(* PLC project  *)

PROGRAM Sensor

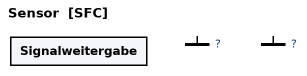
INITIAL_STEP Sensor bereit:
END_STEP
STEP Signalweitergabe:
END_STEP
TRANSITION FROM ? TO ?
  := ?;
END_TRANSITION
TRANSITION FROM ? TO ?
  := ?;
END_TRANSITION
END_PROGRAM
